// TwinCAT 3 PLC project Sample_Vibration
// ProgramVersion: 3.1.4020.10
// libraries:
//   Tc2_Standard, * (Beckhoff Automation GmbH)
//   Tc2_System, * (Beckhoff Automation GmbH)
//   Tc2_Utilities, * (Beckhoff Automation GmbH)
//   Tc3_CM, * (Beckhoff Automation GmbH)
//   Tc3_CM_Base, * (Beckhoff Automation GmbH)
//   Tc3_Module, * (Beckhoff Automation GmbH)
//   Tc3_MultiArray, * (Beckhoff Automation GmbH)
// project tree:
//   DUTs/Error Monitoring/ ST_HRErrHist.TcDUT
//   DUTs/ E_AnalysisIDs.TcDUT, E_IsoClass.TcDUT
//   DUTs/Function Generator/ E_FunctionType.TcDUT (not stored)
//   GVLs/ GVL_Constants.TcGVL
//   / PlcTask.TcTTO, PlcTask_CM.TcTTO
//   POUs/Error Monitoring/ FB_HRErrHist.TcPOU
//   POUs/Function Generator/ FB_FunctionGenerator.TcPOU
//   POUs/ MAIN.TcPOU, MAIN_CM.TcPOU

CONFIGURATION Sample_Vibration
    RESOURCE PLC ON TwinCAT3
        TASK PlcTask(INTERVAL := T#1ms, PRIORITY := 4);
        TASK PlcTask_CM(INTERVAL := T#10ms, PRIORITY := 8);
        PROGRAM MAIN WITH PlcTask : MAIN;
        PROGRAM MAIN_CM WITH PlcTask_CM : MAIN_CM;
    END_RESOURCE
END_CONFIGURATION

// ---- DUTs/Error Monitoring/ST_HRErrHist.TcDUT
TYPE ST_HRErrHist :
STRUCT
{attribute 'displaymode':='hex'}
	hrErrCode	: HRESULT;
	sErrSource	: STRING(63);
	nErrCount	: UDINT;
END_STRUCT
END_TYPE

// ---- DUTs/E_AnalysisIDs.TcDUT
TYPE E_AnalysisIDs :
(
	(* analysis chain *)
	eID_Source := 1,  
	eID_IntRMS,   //  implicitly assigned to 2, which is one greater than the previous value. (automatically increments) Qin
	eID_Sink
) UDINT;
END_TYPE

// ---- DUTs/E_IsoClass.TcDUT
(* ISO Classes *)
{attribute 'qualified_only'}
TYPE E_IsoClass :
(
	A := 1,
	B,
	C,
	D
) UDINT;
END_TYPE

// ---- GVLs/GVL_Constants.TcGVL
VAR_GLOBAL CONSTANT	
	
	cOversamples 	: UDINT 	:= 10;		// number of oversamples
	cFSample        : UDINT     := 10000;   // 1ms task with 10 oversamples = 10kHz
	
	// define FFT parameters, note that cFSample / cWindowLength must be such that numerical frequency resolution
	// is lower than fLowerFrequencyLimit resolution  =  10000/4000 = 2.5 Hz < 10 Hz 
	cFFTLength		: UDINT		:= 4096;	        // length of FFT
    cWindowLength   : UDINT     := 4000;            // 96 samples Zero padding
	cBufferLength	: UDINT		:= cWindowLength/2;	// buffer size due to 50% overlap
	
	// define frequency interval according to ISO 10816-3
	// e.g. 10 .. 1000 Hz for rotating speed over 600r/min
	cfLowerFrequencyLimit : UDINT := 10;   
	cfUpperFrequencyLimit : UDINT := 1000; 
	
	// Parameters for RMS calculation
	cOrderRMS        : UDINT := 2; // ISO 10816-3 requires velocity and displacement, if measured using accelerometer we need to integrate 2 times
	cChannels		 : UDINT := 2; // ISO 10816-3 says 2 orthogonal sensors per measurement location-> 2 channels
	cResult_Length   : UDINT := cOrderRMS+1; // nOrder+1
	
	// Classes according to ISO: machine type 1, stiff location, Class definitions
	cISOClassDef_Velocity  : ARRAY[1..3] OF LREAL := [2.3E-3, 4.5E-3, 7.1E-3];
	cISOClassDef_Displ     : ARRAY[1..3] OF LREAL := [29E-6, 57E-6, 90E-6];	
	
	// optional constants if real sensors are applied
	cGravitationalAcc : LREAL := 9.81;    // 1 g approx 9.81 m/s^2 -> physical constant
	cSensitivity      : LREAL := 0.01;    // [in Volts/g] depends on sensor used in application, e.g. 10 mV/g
	cMeasurementRange : LREAL := 5;       // +-5 Volts (EL3632)
	cResolution       : LREAL := 32768;   // 2^15 (15 bits resolution + 1 bit sign) (EL3632)
	cScale            : LREAL := cMeasurementRange*cGravitationalAcc/(cSensitivity*cResolution);
	
END_VAR

// ---- POUs/MAIN.TcPOU
PROGRAM MAIN
VAR CONSTANT
    cInitSource			: ST_MA_MultiArray_InitPars 
							:= ( eTypeCode := eMA_TypeCode_LREAL, nDims := 2, aDimSizes := [cChannels, cBufferLength]);
	
END_VAR

VAR
	(* Input *)	
	nInputSelection			: UDINT := 1;						// Switch between hardware and function generator	
	nSample					: UDINT;
	// Hardware
	aEl3632Ch1 AT %I*		: ARRAY[1..cOversamples] OF INT;	// Input from hardware e.g. EL3632 ch1
	aEl3632Ch2 AT %I*		: ARRAY[1..cOversamples] OF INT;	// Input from hardware e.g. EL3632 ch2
	// Function generator
	fbFunctionGenerator1	: FB_FunctionGenerator;		// Signal Generator, ch1
	fSetFrequency1			: LREAL := 400;		        // Hz
	fSetAmplitude1			: LREAL := 4;		        // peak amplitude of sin signal [m/s^2]
	fbFunctionGenerator2	: FB_FunctionGenerator;		// Signal Generator, ch2
	fSetFrequency2			: LREAL := 35;		        // Hz
	fSetAmplitude2			: LREAL := 4;		        // peak amplitude of sin signal	[m/s^2]	
		
	
	(* Input from aBuffer to fbSource *)
	aBuffer				: ARRAY[1..cChannels] OF ARRAY[1..cOversamples] OF LREAL;						
	fbSource			: FB_CMA_Source :=(	stInitPars := cInitSource, 
											nOwnID := eID_Source, 
											aDestIDs := [eID_IntRMS]);		// Initialize source buffers
										
	(* From fbSink to aRMSResult *)	
	aRMSResult   		: ARRAY[1..cChannels] OF ARRAY[1..cResult_Length] OF LREAL;	// Copy result									
	fbSink				: FB_CMA_Sink := (nOwnID := eID_Sink);

	
	(* Classify calculated RMS values *)
	nCountResults		  : ULINT;	
	bCalculate			  : BOOL;
	nChannel              : UDINT;
	ISOClassIs_Vel        : ARRAY[1..cChannels] OF E_IsoClass;
	ISOClassIs_Displ      : ARRAY[1..cChannels] OF E_IsoClass;	
	
	(* error monitoring *)
	fbErrHist			: FB_HRErrHist; 

	(* little helper variables *)
	Ch1VelRMS : LREAL;
	Ch1DisplRMS : LREAL;
	Ch2VelRMS : LREAL;
	Ch2DisplRMS : LREAL;	
	
	(* output *)
	ISO_10816_Classification AT%Q* : E_IsoClass;
	
END_VAR

(* Input *)
CASE nInputSelection OF  // switch between 2 data sources --Qin
	0:  (* input from EL3632 *)    // analog input module
		FOR nSample := 1 TO cOversamples DO
			aBuffer[1][nSample] := cScale*INT_TO_LREAL(aEl3632Ch1[nSample]); // convert from Volts to acceleration in m/s^2
			aBuffer[2][nSample] := cScale*INT_TO_LREAL(aEl3632Ch2[nSample]);
		END_FOR 
	1:  (* signal generator *)		// create aritifical sine signal
		fbFunctionGenerator1(	fFrequency 	:= fSetFrequency1,
								fAmplitude 	:= fSetAmplitude1,
								eFunction 	:= E_FunctionType.Sine,
								aSignal		:= aBuffer[1] );	
		fbFunctionGenerator2(	fFrequency 	:= fSetFrequency2,
								fAmplitude 	:= fSetAmplitude2,
								eFunction 	:= E_FunctionType.Sine,
								aSignal		:= aBuffer[2] );	
END_CASE					

(* Call source to collect data *)
fbSource.Input2D( pDataIn 			:= ADR(aBuffer),   // ADR() gets the memory address (pointer). Qin
				  nDataInSize 		:= SIZEOF(aBuffer), 
				  eElementType 		:= eMA_TypeCode_LREAL,
				  nWorkDim0			:= 0,
				  nWorkDim1			:= 1,
				  pStartIndex		:= 0,
				  nOptionPars		:= cCMA_Option_MarkInterruption ); 
				  
IF fbSource.bError THEN
	fbErrHist.AddError(bErr:=TRUE, hrErrCode:=fbSource.hrErrorCode, sErrSource:='MAIN.fbSource'); // error monitoring
	// ToDo: if error
END_IF
(*fbSource is part of TwinCAT's Condition Monitoring & Analytics (CMA) library. It:
Acts as a data input interface for the analytics pipeline
Buffers and manages data flow into processing algorithms
Handles data format conversion and validation
Coordinates with other analytics blocks (like filters, FFT, RMS calculators)*)

(* Push results to sink *)
fbSink.Output2D(	pDataOut 		:= ADR(aRMSResult), 
					nDataOutSize 	:= SIZEOF(aRMSResult), 
					eElementType 	:= eMA_TypeCode_LREAL, 
					nWorkDim0 		:= 0,
					nWorkDim1 		:= 1,
					nElementsDim0	:= 0,
					nElementsDim1	:= 0,
					pStartIndex 	:= 0,
					nOptionPars		:= 0,
					bNewResult		=> bCalculate );
IF fbSink.bError THEN
	fbErrHist.AddError(bErr:=TRUE, hrErrCode:=fbSink.hrErrorCode, sErrSource:='MAIN.fbSink'); // error monitoring
	// ToDo: if error
END_IF

// define class according to ISO 10816-3 based on velocity and displacement data for each measurement channel
IF bCalculate THEN   // Only proceed if fbSink.Output2D(...) has new data. --Qin 
// bCalculate is set to TRUE when fresh results were written into aRMSResult.
	Ch1VelRMS := aRMSResult[1][2];
	Ch1DisplRMS := aRMSResult[1][3];
	Ch2VelRMS := aRMSResult[2][2];
	Ch2DisplRMS := aRMSResult[2][3];	
	
	IF NOT lrealisnan(Ch1VelRMS) THEN 

		nCountResults := fbSink.nCntResults;
		
		// do for each channel
		FOR nChannel := 1 TO cChannels DO
			
			// evaluate velocity data
			ISOClassIs_Vel[nChannel] := E_IsoClass.A;
			IF aRMSResult[nChannel][2] > cISOClassDef_Velocity[3] THEN
				ISOClassIs_Vel[nChannel] := E_IsoClass.D;
			ELSIF aRMSResult[nChannel][2] > cISOClassDef_Velocity[2] THEN
				ISOClassIs_Vel[nChannel] := E_IsoClass.C;
			ELSIF aRMSResult[nChannel][2] > cISOClassDef_Velocity[1] THEN
				ISOClassIs_Vel[nChannel] := E_IsoClass.B;
			END_IF;  
			
			// evaluate displacement data
			ISOClassIs_Displ[nChannel] := E_IsoClass.A;
			IF aRMSResult[nChannel][3] > cISOClassDef_Displ[3] THEN
				ISOClassIs_Displ[nChannel] := E_IsoClass.D;
			ELSIF aRMSResult[nChannel][3] > cISOClassDef_Displ[2] THEN
				ISOClassIs_Displ[nChannel] := E_IsoClass.C;
			ELSIF aRMSResult[nChannel][3] > cISOClassDef_Displ[1] THEN
				ISOClassIs_Displ[nChannel] := E_IsoClass.B;
			END_IF;	
									
		END_FOR;
		
		// according to ISO 10816-3 select worst case 		
		ISO_10816_Classification := E_IsoClass.A;
		FOR  nChannel := 1 TO cChannels DO 
			IF ISOClassIs_Vel[nChannel] >  ISO_10816_Classification THEN
				ISO_10816_Classification := ISOClassIs_Vel[nChannel];
			END_IF
			IF ISOClassIs_Displ[nChannel] >  ISO_10816_Classification THEN
				ISO_10816_Classification := ISOClassIs_Displ[nChannel];
			END_IF
		END_FOR;
	ELSE
		// result is NaN... code here what to do. 
		
	END_IF;
	
END_IF

END_PROGRAM

// ---- POUs/Function Generator/FB_FunctionGenerator.TcPOU
// generates a signal build up by the specified function type. v1.6
FUNCTION_BLOCK FB_FunctionGenerator
VAR_INPUT
	bEnable		: BOOL 	:= TRUE;	// set TRUE to generate the specified signal; set FALSE to reset the signal buffer
	fFrequency	: LREAL := 1000;	// in [Hz]
	fAmplitude	: LREAL := 1;
	fOffset		: LREAL	:= 0;	
	nDutyCycle	: UINT 	:= 50;		// in [%] (for pulse function)
	eFunction	: E_FunctionType := E_FunctionType.Sine;	
END_VAR
VAR_IN_OUT
	aSignal		: ARRAY[1..cOversamples] OF LREAL;
END_VAR
VAR_OUTPUT
	bError		: BOOL;
END_VAR

VAR
	bInit						: BOOL := TRUE;
	fbGetTaskIdx				: GETCURTASKINDEX;
	
	fLastFrequency				: LREAL;		// in [Hz]
	fLastAmplitude				: LREAL;
	fLastOffset					: LREAL;
	nLastDutyCycle				: UINT;
	eLastFunction				: E_FunctionType;
	
	nSamples					: UDINT;
	fCycleTime					: LREAL;		// in [s]
	fDelta						: LREAL;		// amplitude delta per sample
	fPhase						: LREAL;		// in [°]
	nSign						: INT := 1;		// 1 or -1
	fLastSignalValue			: LREAL;		// amplitude
	fPeriod						: LREAL;		// in [s]
	fAngularIncrement			: LREAL;		// in [°]
	fAngularIncrementPerCycle	: LREAL;		// in [°]
	fAngularIncrementPerSample	: LREAL;		// in [°]
	(* for modulated signal (carrier signal without offset) *)
	fCarrierFrequency					: LREAL := 500;	// in [Hz] (sine)
	fCarrierAmplitude					: LREAL := 1;
	fCarrierPeriod						: LREAL;		// in [s]
	fCarrierAngularIncrement			: LREAL;		// in [°]
	fCarrierAngularIncrementPerCycle	: LREAL;		// in [°]
	fCarrierAngularIncrementPerSample	: LREAL;		// in [°]
				
END_VAR

IF bEnable THEN
	IF fLastFrequency <> fFrequency THEN
		bInit := TRUE; // For automatic initializing
		fLastFrequency := fFrequency;
	END_IF
	IF fLastAmplitude <> fAmplitude THEN
		bInit := TRUE; // For automatic initializing
		fLastAmplitude := fAmplitude;
	END_IF
	IF fLastOffset <> fOffset THEN
		bInit := TRUE; // For automatic initializing
		fLastOffset := fOffset;
	END_IF
	IF nLastDutyCycle <> nDutyCycle THEN
		bInit := TRUE; // For automatic initializing
		nLastDutyCycle := nDutyCycle;
	END_IF
	IF eLastFunction <> eFunction THEN
		bInit := TRUE; // For automatic initializing
		eLastFunction := eFunction;
	END_IF
	IF bInit THEN
		// Get task info	
		fbGetTaskIdx();
		fCycleTime := UDINT_TO_LREAL(TwinCAT_SystemInfoVarList._TaskInfo[fbGetTaskIdx.index].CycleTime) (*100ns*) / (10.0 * 1000.0 * 1000.0);	
		fLastSignalValue := 0;
		nSign := 1;
		fAngularIncrement := 0;
		// Flush out old data
		MEMSET(ADR(aSignal), 0, SIZEOF(aSignal));
		IF fFrequency > 0 AND fCycleTime > 0 THEN		
			// Calculate period, increments per plc cycle, increment per oversample
			IF cOversamples > 0 THEN			
				IF eFunction = E_FunctionType.Sine THEN
					fPeriod := 1/fFrequency;
					fAngularIncrementPerCycle := 360*(fCycleTime/fPeriod);
					fAngularIncrementPerSample := fAngularIncrementPerCycle/cOversamples;
					// no phase adjustment
					bInit := FALSE;	
				ELSIF eFunction = E_FunctionType.Square	THEN
					fPeriod := 1/fFrequency;
					fAngularIncrementPerCycle  := 360*(fCycleTime/fPeriod);
					fAngularIncrementPerSample := fAngularIncrementPerCycle/cOversamples;
					fPhase := 0.5*360;
					bInit := FALSE;
				ELSIF eFunction = E_FunctionType.Pulse THEN
					fPeriod := 1/fFrequency;
					fAngularIncrementPerCycle  := 360*(fCycleTime/fPeriod);
					fAngularIncrementPerSample := fAngularIncrementPerCycle/cOversamples;
					IF nDutyCycle > 100 THEN
						nDutyCycle := 100;
					END_IF
					fPhase := (UDINT_TO_LREAL(nDutyCycle)/100)*360;
					bInit := FALSE;					
				ELSIF eFunction = E_FunctionType.Triangular THEN
					fPeriod := 1/fFrequency;				
					fAngularIncrementPerCycle  := 360*(fCycleTime/fPeriod);
					fAngularIncrementPerSample := fAngularIncrementPerCycle/cOversamples;
					fPhase := 0.5*360; 
					fDelta := 4*(fAmplitude/(360/fAngularIncrementPerSample));				
					bInit := FALSE;
				ELSIF eFunction = E_FunctionType.Sawtooth THEN
					fPeriod := 1/fFrequency;			
					fAngularIncrementPerCycle  := 360*(fCycleTime/fPeriod);		
					fAngularIncrementPerSample := fAngularIncrementPerCycle/cOversamples;
					fDelta := fAmplitude/(360/fAngularIncrementPerSample);
					bInit := FALSE;
				ELSIF eFunction = E_FunctionType.AM THEN
					fPeriod := 1/fFrequency;
					fAngularIncrementPerCycle := 360*(fCycleTime/fPeriod);
					fAngularIncrementPerSample := fAngularIncrementPerCycle/cOversamples;
					// no phase adjustment
					fCarrierPeriod := 1/fCarrierFrequency;
					fCarrierAngularIncrementPerCycle := 360*(fCycleTime/fCarrierPeriod);
					fCarrierAngularIncrementPerSample := fCarrierAngularIncrementPerCycle/cOversamples;				
					// no phase adjustment	
					bInit := FALSE;
				ELSE
					bError := TRUE;	
				END_IF
			ELSE
				bError := TRUE;
			END_IF
		ELSE
			bError := TRUE;
		END_IF
	END_IF
	
	// Enable function generator
	IF NOT bError THEN		
		CASE eFunction OF		
			// sine: typical for vibrations originating from rotating machine
			E_FunctionType.Sine: Sine();
			
			// square: mixed sine signals good for analyzing spectrum				
			E_FunctionType.Square: Square();
			
			// pulse: mixed sine signals good for analyzing spectrum				
			E_FunctionType.Pulse: Pulse();
	
			// sawtooth: ramp-type vibrations, continuously increasing			
			E_FunctionType.Sawtooth: Sawtooth();
		
			// triangular: mixed sine signals good for analyzing spectrum
			E_FunctionType.Triangular: Triangular();
		
			// amplitude modulation: typical for vibrations originating from gear-tooth failure or bearing faults
			// Carrier signal with own frequency and amplitude		
			E_FunctionType.AM: AM();				
		END_CASE
	END_IF
ELSE
	// Flush out old data
	MEMSET(ADR(aSignal), 0, SIZEOF(aSignal));    // aSignal is the function block's output array parameter  --Qin
	
	bInit := TRUE;
	bError := FALSE;
END_IF

METHOD PRIVATE AM
VAR_INPUT
END_VAR
{warning disable C0371}

FOR nSamples := 1 TO cOversamples DO
	// base signal * carrier signal
	aSignal[nSamples] := ( fAmplitude*SIN(2*PI*(fAngularIncrement+(nSamples-1)*fAngularIncrementPerSample)/360) + fOffset )
							* ( fCarrierAmplitude*SIN(2*PI*(fCarrierAngularIncrement+(nSamples-1)*fCarrierAngularIncrementPerSample)/360) );
END_FOR
// Increment angular positions
fAngularIncrement := fAngularIncrement + fAngularIncrementPerCycle;
fCarrierAngularIncrement := fCarrierAngularIncrement + fCarrierAngularIncrementPerCycle;

{warning restore C0371}
END_METHOD

METHOD PRIVATE Pulse
VAR_INPUT
END_VAR
{warning disable C0371}

FOR nSamples := 1 TO cOversamples DO
	// For pulse wave (unequal phases)
	IF (fAngularIncrement >= 360) THEN
		fAngularIncrement := fAngularIncrement - DINT_TO_LREAL(LREAL_TO_DINT(fAngularIncrement/360))*360;
		// or with Tc2_Math library: fAngularIncrement := LMOD(fAngularIncrement,360);
	END_IF
	IF (fAngularIncrement < fPhase) THEN
		nSign := 1;		
	ELSIF (fAngularIncrement >= fPhase) THEN
		nSign := 0;
	END_IF
	fAngularIncrement := fAngularIncrement + fAngularIncrementPerSample;
	
	aSignal[nSamples] := nSign*fAmplitude;
	
	aSignal[nSamples] := aSignal[nSamples] + fOffset;
END_FOR

{warning restore C0371}
END_METHOD

METHOD PRIVATE Sawtooth
VAR_INPUT
END_VAR
{warning disable C0371}

FOR nSamples := 1 TO cOversamples DO
	// For sawtooth wave (equal phase = period/2)
	IF (fAngularIncrement >= 360) THEN
		fAngularIncrement := fAngularIncrement - DINT_TO_LREAL(LREAL_TO_DINT(fAngularIncrement/360))*360;
		// or with Tc2_Math library: fAngularIncrement := LMOD(fAngularIncrement,360);
		fLastSignalValue := fLastSignalValue -fAmplitude;
	END_IF
	fAngularIncrement := fAngularIncrement + fAngularIncrementPerSample;

	aSignal[nSamples] := fLastSignalValue + fDelta;

	// Store last sample
	fLastSignalValue := aSignal[nSamples];
	
	aSignal[nSamples] := aSignal[nSamples] + fOffset;					
END_FOR	

{warning restore C0371}
END_METHOD

METHOD PRIVATE Sine
VAR_INPUT
END_VAR
{warning disable C0371}

FOR nSamples := 1 TO cOversamples DO
	aSignal[nSamples] := fAmplitude*SIN(2*PI*(fAngularIncrement+(nSamples-1)*fAngularIncrementPerSample)/360);

	aSignal[nSamples] := aSignal[nSamples] + fOffset;
END_FOR

// Increment angular position
fAngularIncrement := fAngularIncrement + fAngularIncrementPerCycle;

{warning restore C0371}
END_METHOD

METHOD PRIVATE Square
VAR_INPUT
END_VAR
{warning disable C0371}

FOR nSamples := 1 TO cOversamples DO
	// For square wave (equal phase = period/2)
	IF (fAngularIncrement >= 360) THEN
		fAngularIncrement := fAngularIncrement - DINT_TO_LREAL(LREAL_TO_DINT(fAngularIncrement/360))*360;
		// or with Tc2_Math library: fAngularIncrement := LMOD(fAngularIncrement,360);
	END_IF
	IF (fAngularIncrement < fPhase) THEN
		nSign := 1;
	ELSIF (fAngularIncrement >= fPhase) THEN
		nSign := -1;
	END_IF
	fAngularIncrement := fAngularIncrement + fAngularIncrementPerSample;
	
	aSignal[nSamples] := nSign*fAmplitude;
	
	aSignal[nSamples] := aSignal[nSamples] + fOffset;
END_FOR

{warning restore C0371}
END_METHOD

METHOD PRIVATE Triangular
VAR_INPUT
END_VAR
{warning disable C0371}

FOR nSamples := 1 TO cOversamples DO
	IF (fAngularIncrement >= 360) THEN
		fAngularIncrement := fAngularIncrement - DINT_TO_LREAL(LREAL_TO_DINT(fAngularIncrement/360))*360;
		// or with Tc2_Math library: fAngularIncrement := LMOD(fAngularIncrement,360);
	END_IF
	// Negative delta -> Positive delta
	IF fAngularIncrement < fPhase/2 THEN	
		nSign := 1;		
	ELSIF fAngularIncrement >= fPhase/2 AND fAngularIncrement < 3*fPhase/2 THEN
		nSign := -1;
	ELSIF fAngularIncrement >= 3*fPhase/2 THEN
		nSign := 1;	
	END_IF
	fAngularIncrement := fAngularIncrement + fAngularIncrementPerSample;
	
	aSignal[nSamples] := fLastSignalValue + nSign*fDelta;
	IF aSignal[nSamples] > fAmplitude THEN
		aSignal[nSamples] := aSignal[nSamples] - 2*(aSignal[nSamples]-fAmplitude);
	ELSIF aSignal[nSamples] < (-1)*fAmplitude THEN
		aSignal[nSamples] := aSignal[nSamples] - 2*(aSignal[nSamples]+fAmplitude);
	END_IF
	
	// Store last sample
	fLastSignalValue := aSignal[nSamples];		
	
	aSignal[nSamples] := aSignal[nSamples] + fOffset;
END_FOR

{warning restore C0371}
END_METHOD

END_FUNCTION_BLOCK

// ---- POUs/Error Monitoring/FB_HRErrHist.TcPOU
FUNCTION_BLOCK FB_HRErrHist
(* v1.10
build up an error history consisting of two arrays and one index.
The index shows the actual array position. The last error id and the count for this id are saved in the arrays.
If an error id is the same as the previous input error the counter is increased. Otherwise the index is increased.
*)
VAR_INPUT
	bEdgeDetect	: BOOL;	(* FALSE: every input(bErr) is processed; TRUE: only rising edge of input is processed *)
END_VAR
VAR_OUTPUT
	nErrSum		: UINT;
	nErrIdx		: UINT; // error list index of last occured error (max. cHistLen)
	aErrList	: ARRAY[1..cHistLen] OF ST_HRErrHist;
END_VAR

VAR
	bNewErr		: BOOL;
	fbErrTrig	: R_TRIG;
END_VAR
VAR CONSTANT
	cHistLen	: UINT := 100;
END_VAR

METHOD AddError
VAR_INPUT
	bErr		: BOOL;
	hrErrCode	: HRESULT;
	sErrSource	: STRING(63);
END_VAR
fbErrTrig(CLK:=bErr);
IF bEdgeDetect THEN
	bNewErr := fbErrTrig.Q;
ELSE
	bNewErr := bErr;
END_IF

IF bNewErr THEN
	nErrSum := nErrSum + 1;
	IF nErrIdx < cHistLen THEN
		IF nErrIdx = 0 THEN
			nErrIdx	:= nErrIdx + 1;
		ELSIF aErrList[nErrIdx].hrErrCode <> hrErrCode OR aErrList[nErrIdx].sErrSource <> sErrSource THEN
			nErrIdx	:= nErrIdx + 1;
		END_IF
		aErrList[nErrIdx].hrErrCode := hrErrCode;
		aErrList[nErrIdx].sErrSource := sErrSource;
		aErrList[nErrIdx].nErrCount := aErrList[nErrIdx].nErrCount + 1;
	END_IF
END_IF
END_METHOD

METHOD Reset
VAR_INPUT
END_VAR
nErrSum := 0;
nErrIdx := 0;
MEMSET(ADR(aErrList),0,SIZEOF(aErrList));
END_METHOD

END_FUNCTION_BLOCK

// ---- POUs/MAIN_CM.TcPOU
PROGRAM MAIN_CM
VAR CONSTANT
	cInitIntRMS 	: ST_CM_IntegratedRMS_InitPars   := (	nFFT_Length := cFFTLength, 
															nWindowLength := cWindowLength,
															fSampleRate := cFSample,
		 													fLowerFrequencyLimit := cfLowerFrequencyLimit,
															fUpperFrequencyLimit := cfUpperFrequencyLimit,
															nOrder := cOrderRMS,
															nChannels := cChannels,                        
															eWindowType := E_CM_WindowType.eCM_HannWindow, 
															bTransformToDecibel:= FALSE);								
END_VAR

VAR	
	fbRMS				: FB_CMA_IntegratedRMS  	  :=(	stInitPars := cInitIntRMS, 
															nOwnID := eID_IntRMS, 
															aDestIDs := [eID_Sink] );

	fbErrHist			: FB_HRErrHist; // error monitoring

END_VAR

// Call RMS
fbRMS.Call();
IF fbRMS.bError THEN
	fbErrHist.AddError(bErr:=TRUE, hrErrCode:=fbRMS.hrErrorCode, sErrSource:='MAIN_CM.fbRMS'); // error monitoring
	// ToDo: if error
END_IF

END_PROGRAM
